FUNCTION_BLOCK  TcoFeedingSequenceTask EXTENDS TcoCore.TcoTask
VAR_IN_OUT
	inoStatus:TcoFeeding_Status_v_1_x_x;
	inoConfig:TcoFeeding_Config_v_1_x_x;

END_VAR
VAR
	_sequence      : TcoCore.TcoSequence(THIS^, eRestoreMode.None);
    _observerSequence       : TcoCore.TcoSequencerObserver(THIS^);
	_infoTime:TIME;
	_errorTime:	TIME;
	_errorMessage:TcoCore.TcoMessenger(THIS^);

END_VAR

IF  __ISVALIDREF(inoConfig) THEN  
_infoTime := THIS^.inoConfig.InfoTime;
_errorTime := THIS^.inoConfig.ErrorTime;
END_IF;

PROPERTY PUBLIC ErrorTime : REFERENCE TO TIME
GET
ErrorTime REF=_errorTime;
END_GET
END_PROPERTY

METHOD PUBLIC HandleTaskError :BOOL;
VAR_INPUT
END_VAR
IF THIS^.ElapsedTime > THIS^.ErrorTime AND THIS^.ErrorTime<>T#0S THEN
	THIS^.ThrowWhen(TRUE);
END_IF

HandleTaskError := THIS^.Error AND NOT THIS^._errorMessage.Pinned;
END_METHOD

PROPERTY InfoTime :REFERENCE TO TIME
GET
InfoTime REF=_infoTime;
END_GET
END_PROPERTY

PROPERTY PUBLIC Observer : REFERENCE TO TcoCore.TcoSequencerObserver
GET
Observer ref=_observerSequence;
END_GET
END_PROPERTY

METHOD PROTECTED OnError
VAR
	description: STRING;
END_VAR
description := '<#Task finished with error.#>'; 
IF  __ISVALIDREF(inoStatus) THEN   THIS^.inoStatus.ActionDescription := description; END_IF;
THIS^._errorMessage.Error('To restore acknowledge this alarm.').Pin();
END_METHOD

(*~
	<docu>
		<summary>
			Restores this instance to the Ready state. Can be called explicitly or from within one of the restore mechanisms.
			<para>
				See also <see cref="PlcDocu.TcoCore.TcoTask.AutoRestorable()"/>
			</para>
		</summary>			
	</docu>	
~*)
METHOD Restore : ITcoRestorable
SUPER^.Restore();
_sequence.ModeController.Mode :=eSequencerMode.CyclicMode;
_messenger.UnPin();
_errorMessage.UnPin();
_sequence.Restore();
END_METHOD

PROPERTY PUBLIC Sequence : REFERENCE TO TcoCore.TcoSequence
GET
Sequence ref=_sequence;
END_GET
END_PROPERTY

METHOD SetCyclicMode
VAR_INPUT
END_VAR
_sequence.ModeController.Mode :=eSequencerMode.CyclicMode;
END_METHOD

METHOD SetStepMode
VAR_INPUT
END_VAR
_sequence.ModeController.Mode :=eSequencerMode.StepMode;
END_METHOD

END_FUNCTION_BLOCK

(* stored: Version 1.1.0.1
   POU TcoFeedingSequenceTask: Id {6a15bf14-7b1b-4cbd-8547-7cf38af9c488}, SpecialFunc None
   Property ErrorTime: Id {05e1ad56-dadc-4374-87ee-8893b1532d45}
   Get Get: Id {cf0c7697-f2bd-4496-a450-d4f32e0dcce0}
   Method HandleTaskError: Id {79e1455e-3b62-4778-9ae8-b65f29dd5ccc}
   Property InfoTime: Id {b3b0b370-1c03-46ec-989c-044a8dcfd7e3}
   Get Get: Id {9018b3b8-6b97-4ff3-9498-2731bd542746}
   Property Observer: Id {9113932a-5f79-4cb8-913e-f1f163042dcd}
   Get Get: Id {2c81941f-30e5-4583-aacb-87ec3829c12b}
   Method OnError: Id {e7b2d8c9-4a9f-4d08-8aa2-c09fc50ea9c7}
   Method Restore: Id {70622ba5-65b1-4df5-a40b-3f44610a5cf5}
   Property Sequence: Id {94bbc59b-0664-426f-bfe4-95dc7aefb9fd}
   Get Get: Id {ac4daf50-fcf1-445e-abd1-05fe37c35ab0}
   Method SetCyclicMode: Id {d8d44d3b-7673-4c73-9e75-69b113838d72}
   Method SetStepMode: Id {f61443ff-a06e-4b18-927e-d9bc6fb09bfc} *)
